// TwinCAT 3 PLC project VCM_lib
// Title: Twincat 3 Tutorial
// Company: MyAutomation MA-IT
// Author: S. Klaver
// ProjectVersion: 1.1.0
// Description: This is a librarry tutorial project
// libraries:
//   Tc2_Standard, * (Beckhoff Automation GmbH)
//   Tc2_System, * (Beckhoff Automation GmbH)
//   Tc3_Module, * (Beckhoff Automation GmbH)
//   Twincat 3 Tutorial, * (MA-IT)
//   VisuSymbols,3.5.10.0,System
// project tree:
//   DUTs/ DUT_ALM.TcDUT, DUT_Control_Base.TcDUT, DUT_CS.TcDUT, DUT_HMI.TcDUT, DUT_IO.TcDUT, DUT_STS.TcDUT, DUT_VALVE.TcDUT
//   / GlobalTextList.TcGTLO
//   GVLs/ GVL_VCM.TcGVL
//   POUs/ FB_Valve_monostable.TcPOU, MAIN.TcPOU
//   POUs/Utilities/ FB_DUT_HMI.TcPOU, FB_Integer_To_BooleanArray.TcPOU
//   VISUs/ Main_Visu.TcVIS, ValveHMI.TcVIS
// (motion and I/O tree: see PLC project vcm)
// real-time tasks:
//   TASK PlcTask: cycle T#10ms, priority 20, ADS port 350
//   TASK VISU_TASK: cycle T#200000us, priority 30, ADS port 351

// ---- DUTs/DUT_ALM.TcDUT
TYPE DUT_ALM :
STRUCT
	GeneralFailure: BOOL;
	TimeFailure: BOOL;
	InAlarm: BOOL := TimeFailure OR GeneralFailure;
END_STRUCT
END_TYPE

// ---- DUTs/DUT_Control_Base.TcDUT
TYPE DUT_Control_Base :
STRUCT
	Open :BOOL;
	Close :BOOL;
	Reset :BOOL;
	Simulation :BOOL;
	AutoOn :BOOL;
	AutoOff :BOOL;
	ManualOn :BOOL;
	ManualOff :BOOL;
END_STRUCT
END_TYPE

// ---- DUTs/DUT_CS.TcDUT
TYPE DUT_CS EXTENDS DUT_Control_Base :
STRUCT
	Auto :BOOL;
	Manual :BOOL;
    Interlock :BOOL;
END_STRUCT
END_TYPE

// ---- DUTs/DUT_HMI.TcDUT
TYPE DUT_HMI EXTENDS DUT_Control_Base :
STRUCT
	ModeValue : INT:= 1; // 0: Manual; 1: Auto;
	DisableAutoManual : BOOL;
END_STRUCT
END_TYPE

// ---- DUTs/DUT_IO.TcDUT
TYPE DUT_IO :
STRUCT
	I_isOpen: BOOL := FALSE;
	I_isClosed: BOOL := FALSE;
	I_hasFailure: BOOL := FALSE;
	O_setOpen: BOOL := FALSE;
END_STRUCT
END_TYPE

// ---- DUTs/DUT_STS.TcDUT
TYPE DUT_STS :
STRUCT
	State : INT;
	ManualMode: BOOL;
	AutoMode: BOOL := TRUE;
	InSimulation: BOOL;
	Closed: BOOL := TRUE;
	Opening: BOOL;
	Open: BOOL:= TRUE;
	Closing: BOOL;
	Interlock: BOOL;
	Alarm: BOOL;
END_STRUCT	
	
END_TYPE

// ---- DUTs/DUT_VALVE.TcDUT
TYPE DUT_VALVE :
STRUCT
	Cs: DUT_CS;
	Hmi: DUT_HMI;
	Sts: DUT_STS;
	Alm: DUT_ALM;
	TagName: STRING := '###';
END_STRUCT
END_TYPE

// ---- GVLs/GVL_VCM.TcGVL
{attribute 'qualified_only'}
VAR_GLOBAL
	valve01: DUT_VALVE;
	ioValve01: DUT_IO;
	valve02: DUT_VALVE;
	ioValve02: DUT_IO;
END_VAR

VAR_GLOBAL CONSTANT
	STS_UNDEFINED : INT := 0;
	STS_CLOSED : INT := 10;
	STS_OPENING : INT := 20;
	STS_OPEN : INT := 30;
	STS_CLOSING : INT := 40;
END_VAR

// ---- POUs/FB_Valve_monostable.TcPOU
FUNCTION_BLOCK FB_Valve_monostable
VAR_INPUT
	MaxOpenCloseDuration: INT; //(s) Maximum time the valve needs to open or close in seconds
END_VAR
VAR_OUTPUT
	setOpen: BOOL;
END_VAR
VAR_IN_OUT
	Valve: DUT_VALVE;
	I_O: DUT_IO;
END_VAR
VAR
	openingTimer: Tc2_Standard.TON;
	closingTimer: Tc2_Standard.TON;
	fbHmiDut: FB_DUT_HMI; 
	manualOpen: BOOL;
	manualClose: BOOL;
	manualReset: BOOL;
	reqOpen: BOOL;
	reqClose: BOOL;
	isOpen: BOOL;
	isClosed: BOOL;
	startOpeningTimeOut: BOOL;
	startClosingTimeOut: BOOL;
	fbDutHmi: FB_DUT_HMI;
	
END_VAR

{region Input} 
//set INTERNAL variables
// hmi-open command
IF Valve.Hmi.Open THEN
	manualOpen := TRUE;
	Valve.Hmi.Open := FALSE;
END_IF

// hmi-close command
IF Valve.Hmi.Close THEN
	manualClose := TRUE;
	Valve.Hmi.Close := FALSE;
END_IF

// manual_reset command
IF Valve.Hmi.Reset OR manualReset THEN
	manualReset := TRUE;
	Valve.Hmi.Reset := FALSE;
END_IF 			

// Created Utitlities FB's for learning, can also use altenative (simplefied) code here  
// tried to avoid redunant (HMI) logic.
fbDutHmi(hmiValue_in:= Valve.Hmi);
Valve.Hmi := fbDutHmi.hmiValue_out;
	 
//Set HMI modus overide HMI by CS
Valve.Hmi.DisableAutoManual := Valve.Cs.ManualOn OR Valve.Cs.AutoOn;
IF Valve.Cs.ManualOn THEN
	Valve.Hmi.ManualOn := TRUE;
	Valve.Hmi.ManualOff := FALSE;
	Valve.Hmi.AutoOn := FALSE;
	Valve.Hmi.AutoOff := FALSE;
	Valve.Hmi.ModeValue := 0;
END_IF

IF Valve.Cs.AutoOn THEN
	Valve.Hmi.ManualOn := FALSE;
	Valve.Hmi.ManualOff := FALSE;
	Valve.Hmi.AutoOn := TRUE;
	Valve.Hmi.AutoOff := FALSE;
	Valve.Hmi.ModeValue := 1;
END_IF
	  
{endregion input}
	 

{region interlock-manual-auto}
Valve.Sts.InSimulation := Valve.Cs.Simulation OR Valve.Hmi.Simulation; 
Valve.Sts.Interlock := Valve.Cs.Interlock;

// Set Auto/Manual mode
// CS is Dominant over HMI
Valve.Sts.ManualMode S= (Valve.Cs.Manual OR Valve.Hmi.ManualOn) AND NOT(Valve.Cs.Auto);
Valve.Sts.ManualMode R= (Valve.Cs.Auto OR Valve.Hmi.AutoOn) AND NOT(Valve.Cs.Manual);
Valve.Sts.AutoMode:= NOT(Valve.Sts.ManualMode);
{endregion interlock manual auto}

{region control coördination} 
              
// determine the actual or required state
reqOpen S= (Valve.Sts.AutoMode AND Valve.Cs.Open) OR (Valve.Sts.ManualMode AND manualOpen);
reqOpen R= isOpen;
reqClose S= Valve.Sts.Interlock OR (Valve.Sts.AutoMode AND Valve.Cs.Close) OR (Valve.Sts.ManualMode AND manualClose);
reqClose R= isClosed;
isOpen S= I_O.I_isOpen OR (Valve.Sts.InSimulation AND reqOpen);
isOpen R= NOT (I_O.I_isOpen);	 
isClosed S= I_O.I_isClosed OR (Valve.Sts.InSimulation AND reqClose);
isClosed R= NOT (I_O.I_isClosed);

// set state
IF reqClose THEN
    Valve.Sts.State := GVL_VCM.STS_CLOSING;
ELSIF reqOpen THEN
    Valve.Sts.State := GVL_VCM.STS_OPENING;
ELSIF isOpen THEN
    Valve.Sts.State := GVL_VCM.STS_OPEN;
ELSIF isClosed THEN
    Valve.Sts.State := GVL_VCM.STS_CLOSED;


END_IF

// INIT STS.State zet to CLOSING if UNDEFINED
IF Valve.Sts.State = GVL_VCM.STS_UNDEFINED THEN
	Valve.Sts.State := GVL_VCM.STS_CLOSING;		 
END_IF
		  
CASE Valve.Sts.State OF
    10: //isClosed
        Valve.Sts.Closed := TRUE;
        Valve.Sts.Opening := FALSE;
        Valve.Sts.Open := FALSE;
        Valve.Sts.Closing := FALSE;
    20: //opening
        Valve.Sts.Closed := FALSE;
        Valve.Sts.Opening := TRUE;
        Valve.Sts.Open := FALSE;
        Valve.Sts.Closing := FALSE;
    30: // isOpen
        Valve.Sts.Closed := FALSE;
        Valve.Sts.Opening := FALSE;
        Valve.Sts.Open := TRUE;
        Valve.Sts.Closing := FALSE;
    40: // closing
        Valve.Sts.Closed := FALSE;
        Valve.Sts.Opening := FALSE;
        Valve.Sts.Open := FALSE;
        Valve.Sts.Closing := TRUE;
END_CASE

{endregion}

{region set timer guard for opening and closing}
// Don't use the same timer for opening or closing in case opening or closing is called while previous opening or closing action isn't finished yet.
// Can only be done if a 'DirectionChanged' variable is used. 
//opening timeout guard
startOpeningTimeOut S= NOT (Valve.Sts.Interlock) AND Valve.Sts.Opening;
startOpeningTimeOut R= Valve.Sts.Open OR Valve.Sts.Closing;
openingTimer(IN := startOpeningTimeOut, PT:= INT_TO_TIME(MaxOpenCloseDuration * 1000));
//closing timeout guard
startClosingTimeOut S= Valve.Sts.Interlock OR Valve.Sts.Closing;
startClosingTimeOut R= Valve.Sts.Closed OR Valve.Sts.Opening;
closingTimer(IN := startClosingTimeOut, PT:= INT_TO_TIME(MaxOpenCloseDuration * 1000));

{endregion}

{region Handle alarms}
IF Valve.Cs.Reset OR manualReset THEN
	//reset inAlarm only demand
    Valve.Alm.InAlarm := FALSE;
END_IF
// check if failure (still) exist.
Valve.Alm.TimeFailure := openingTimer.Q OR closingTimer.Q; // Set TimeFailure on opening or closing timeOut
Valve.Alm.GeneralFailure := I_O.I_hasFailure; // Set GeneralFailure
Valve.Alm.InAlarm := Valve.Alm.GeneralFailure OR Valve.Alm.TimeFailure OR Valve.Alm.InAlarm;
{endregion}

{region outputs}
// set/reset output (O_setOpen)
I_O.O_setOpen S= (Valve.Sts.Opening OR Valve.Sts.Open); //Warning: Valve is monostable, keep output also open on status: Valve.Sts.Open
I_O.O_setOpen R= Valve.Sts.Closing OR Valve.Sts.Interlock OR Valve.Sts.InSimulation;

{endregion}

{region cleanup state}
	manualClose R= TRUE;
	manualOpen R= TRUE;
	manualReset R= TRUE;
{endregion}

END_FUNCTION_BLOCK

// ---- POUs/Utilities/FB_DUT_HMI.TcPOU
FUNCTION_BLOCK PUBLIC FB_DUT_HMI
VAR_INPUT
END_VAR
VAR_INPUT
    hmiValue_in: DUT_HMI;
END_VAR
VAR_OUTPUT
    hmiValue_out: DUT_HMI;
END_VAR
VAR
    intToBool: FB_Integer_To_BooleanArray;
    rbModeValues : ARRAY[0..1] OF BOOL;
	i: INT;
	ArrayLength: INT;
	OutputValue: INT;
	IntegerValue: INT;
END_VAR


//Convert HMI radioButton to BOOL
intToBool(IntegerValue:= hmiValue_in.ModeValue, ArrayLength:= 2);
hmiValue_out := hmiValue_in;
// Use BOOL array to set DUT_HMI values
rbModeValues := intToBool.OutputValue;	 
hmiValue_out.ManualOn := rbModeValues[0];
hmiValue_out.ManualOff := NOT rbModeValues[0];
hmiValue_out.AutoOn := rbModeValues[1];
hmiValue_out.AutoOff := NOT rbModeValues[1];

END_FUNCTION_BLOCK

// ---- POUs/Utilities/FB_Integer_To_BooleanArray.TcPOU
FUNCTION_BLOCK FB_Integer_To_BooleanArray
VAR_INPUT
	IntegerValue: INT := -1; // Inte value from Radiobutoon or whatever indexed component
	ArrayLength: INT := 2; // rquired length of the output Array 
END_VAR
VAR_OUTPUT
	OutputValue: ARRAY [0..1] OF BOOL; 
END_VAR
VAR
	i: INT;  // Loop counter
END_VAR

END_FUNCTION_BLOCK

// ---- POUs/MAIN.TcPOU
PROGRAM MAIN
VAR
	isFirstStart : BOOL := TRUE;
	valve_01 : FB_Valve_monostable;
	valve_02 : FB_Valve_monostable;
	
END_VAR

// Set IN(IT)
valve_01.MaxOpenCloseDuration := 180;// this setting can be reduced during test without the fysical Valve
valve_02.MaxOpenCloseDuration := 10;
GVL_VCM.valve01.TagName := 'Valve-01';
GVL_VCM.valve02.TagName := 'Valve-02';

IF isFirstStart THEN
	// Init the Valve at startup (for test/demo)
	GVL_VCM.ioValve01.I_isClosed := TRUE;
	GVL_VCM.ioValve02.I_isClosed := TRUE;
END_IF

// Do stuff
//create valve-01
valve_01(Valve:= GVL_VCM.valve01, I_O:= GVL_VCM.ioValve01);
//create valve-02
valve_02(Valve:= GVL_VCM.valve02, I_O:= GVL_VCM.ioValve02);

isFirstStart := FALSE;

END_PROGRAM

// ---- GlobalTextList.TcGTLO
TEXTLIST GlobalTextList
  204 = '%b'
  80 = '%d'
  37 = '%s'
  224 = '??'
  555 = 'Alarm'
  627 = 'Auto'
  396 = 'Close Valve'
  865 = 'CS Interlock'
  570 = 'CS,Manual'
  936 = 'CS.Auto'
  283 = 'CS.AutoOff'
  660 = 'CS.AutoOn'
  562 = 'CS.Close'
  672 = 'CS.Interlock'
  623 = 'CS.Manual'
  486 = 'CS.ManualOff'
  454 = 'CS.ManualOn'
  384 = 'CS.Off'
  279 = 'CS.On'
  817 = 'CS.OPen'
  138 = 'CS.Open'
  376 = 'CS.Reset'
  512 = 'CS.ResetOff'
  97 = 'CS.ResetOn'
  130 = 'CS.Simulation'
  929 = 'dsfdsf'
  687 = 'en dit?'
  585 = 'GroupBox'
  725 = 'ik ben analoog'
  491 = 'ik ben de tooltip'
  847 = 'Ik ben een schakelaar'
  72 = 'Ik zeg iets over de schakelaar'
  628 = 'Interlock'
  837 = 'Interlocked'
  331 = 'io_values.O_setOpen'
  46 = 'I_hasFailure'
  904 = 'I_isClosed'
  233 = 'I_isOpen'
  182 = 'I_setOpen'
  626 = 'Manual'
  650 = 'None'
  36 = 'Only for Demo and testing'
  352 = 'Open Valve'
  610 = 'O_setOpen'
  954 = 'Reset'
  371 = 'SIM I_hasFailure'
  899 = 'SIM I_IO.hasFailure'
  293 = 'Sim I_IO.isClosed'
  885 = 'SIM I_IO>hasFailure'
  684 = 'Sim I_isClosed'
  444 = 'Simulation'
  822 = 'Sim_IO.isOpen'
  125 = 'Sim_isOpen'
  586 = 'State'
  475 = 'STS'
  937 = 'STS.Open '
  821 = 'STS.State'
  408 = 'Tag'
  934 = 'Tag: {Valve.TagName}'
  109 = 'Temporary for Demo and testing'
  946 = 'Temporary Only for Demo and testing'
  569 = 'tooltip tekst tester'
  50 = 'Valve ##'
  350 = 'Valve ## (FDS assignment)'
  170 = 'Valve (monostable)'
  577 = 'Valve 01'
  844 = 'Valve Control'
  909 = 'Valve FDS assignment'
  724 = 'Valve Mode'
  387 = 'werkt dit?'
  14 = 'zichtbaar?'
  685 = '{Valve.TagName}'
  380 = '{Valve.TagName} - ??'
END_TEXTLIST

// ---- VISUs/Main_Visu.TcVIS
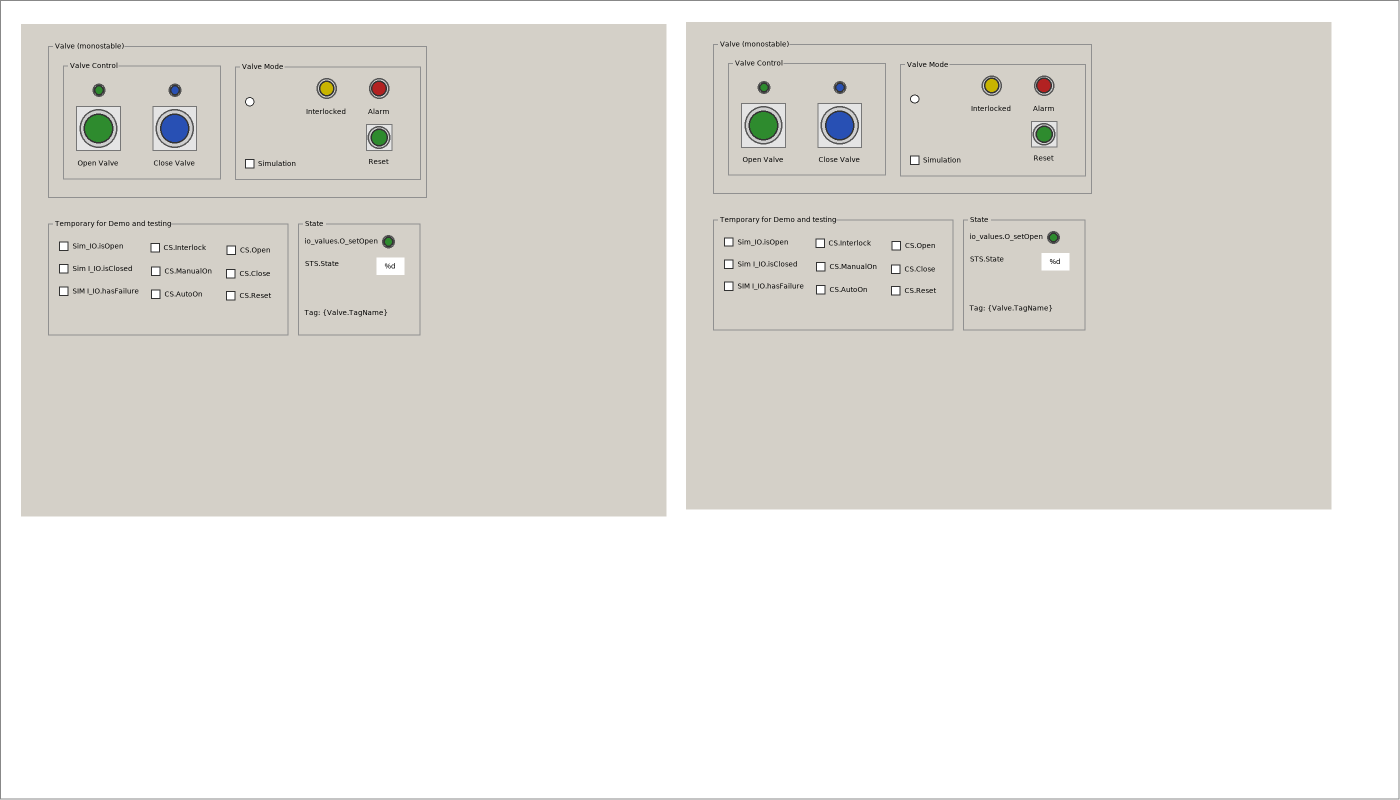
VISUALIZATION Main_Visu  // 1400x800
    Frame (21,24 645x492)
        shows ValveHMI(Valve := GVL_VCM.valve01)
        shows ValveHMI(Valve := GVL_VCM.valve01, ValveIO := GVL_VCM.ioValve01)
    Frame (686,22 645x487)
        shows ValveHMI(Valve := GVL_VCM.valve02, ValveIO := GVL_VCM.ioValve02)
END_VISUALIZATION

// ---- VISUs/ValveHMI.TcVIS
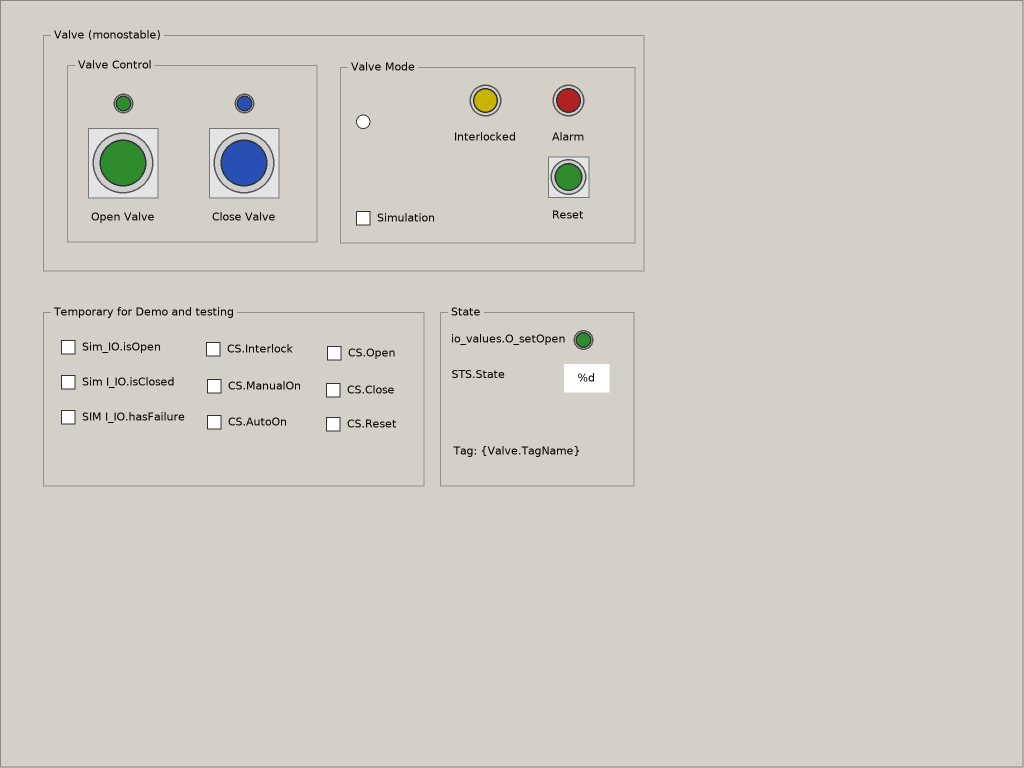
VISUALIZATION ValveHMI  // 1024x768
VAR_IN_OUT
	Valve: DUT_VALVE;
	ValveIO: DUT_IO;
END_VAR
    GroupBox (43,27 601x244), "Valve (monostable)"
        GroupBox (24,30 250x185), "Valve Control"
            PushSwitch (21,71 70x70), variable: Valve.Hmi.Open, behaviour: TOGGLE, style: Switch-PushSwitch-Green
            Lamp1 (45,35 23x23), variable: Valve.Sts.Open, style: Lamp-Lamp1-Green
            Label (14,145 84x30), "Open Valve"
            PushSwitch (142,71 70x70), variable: Valve.Hmi.Close, behaviour: TOGGLE, style: Switch-PushSwitch-Blue
            Label (135,145 84x30), "Close Valve"
            Lamp1 (166,35 23x23), variable: Valve.Sts.Closed, style: Lamp-Lamp1-Blue
        GroupBox (297,32 295x184), "Valve Mode"
            Lamp1 (210,22 37x39), variable: Valve.Alm.InAlarm, style: Lamp-Lamp1-Red
            Label (186,63 84x30), "Alarm"
            RadioButton (14,29 96x67), variable: Valve.Hmi.ModeValue, input disabled if: Valve.Hmi.DisableAutoManual
                Areas[0]: Text=Radiobutton
                Areas[1]: Text=Radiobutton
                p340057476: Manual
                p3123465237: Auto
                p2481256679: Interlock
            PushSwitch (208,93 41x50), variable: Valve.Hmi.Reset, behaviour: TOGGLE, style: Switch-PushSwitch-Green
            Label (186,141 84x30), "Reset"
            Label (103,63 84x30), "Interlocked"
            Lamp1 (127,22 37x39), variable: Valve.Sts.Interlock, style: Lamp-Lamp1-Yellow
            Checkbox (14,144 150x30), "Simulation", variable: Valve.Hmi.Simulation
    GroupBox (43,304 381x182), "Temporary for Demo and testing"
        Checkbox (16,28 133x30), "Sim_IO.isOpen", variable: ValveIO.I_isOpen
        Checkbox (16,63 133x30), "Sim I_IO.isClosed", variable: ValveIO.I_isClosed
        Checkbox (16,98 143x30), "SIM I_IO.hasFailure", variable: ValveIO.I_hasFailure
        Checkbox (161,30 109x30), "CS.Interlock", variable: Valve.Cs.Interlock
        Checkbox (162,67 120x30), "CS.ManualOn", variable: Valve.Cs.ManualOn
        Checkbox (162,103 109x30), "CS.AutoOn", variable: Valve.Cs.AutoOn
        Checkbox (281,71 95x30), "CS.Close", variable: Valve.Cs.Close
        Checkbox (282,34 93x30), "CS.Open", variable: Valve.Cs.Open
        Checkbox (281,105 95x30), "CS.Reset", variable: Valve.Cs.Reset
    GroupBox (440,304 194x182), "State"
        Lamp1 (132,24 23x24), variable: ValveIO.O_setOpen, style: Lamp-Lamp1-Green
        Label (2,20 133x30), "io_values.O_setOpen"
        Label (74,91 53x30)
        Label (4,57 69x27), "STS.State"
        Textfield (123,59 47x30), "%d", text variable: Valve.Sts.State
        Label (2,132 150x30), "Tag: {Valve.TagName}"
END_VISUALIZATION
